FUNCTION alg_a_x2testing : BOOL
VAR_INPUT
	state: STATE;
END_VAR

alg_a_x2testing := state.dvar_M_example_controller_a_x2testing;

END_FUNCTION

(* stored: Version 1.1.0.1, ProductVersion 3.1.4022.18
   POU alg_a_x2testing: Id {dbc56d6a-cf30-41ba-974d-7b5b44af30b9}, SpecialFunc None *)
